Universal Robots PolyScope program: test2.v2objects.urp

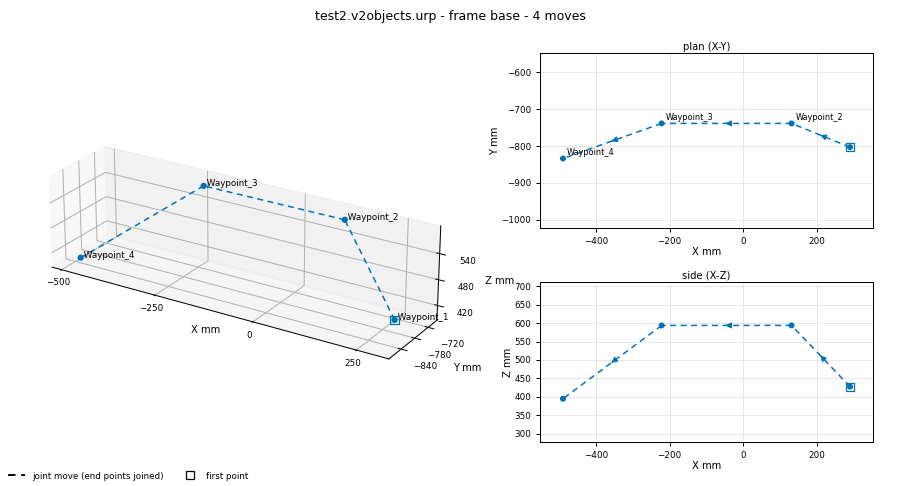
[picture p0: tool path of test2.v2objects.urp in frame base, 4 of 4 moves have a stored position in this frame; points joined in program order, loops and branches not executed]
Program test2.v2objects (installation=default directory=/programs/usbdisk/test 2_v2 createdIn=5.11.10.1010502 lastSavedIn=5.11.10.1010502 robotSerialNumber=20225201357)
Calibrated DH parameters: a=[-0.000097, -0.065329, -0.560646, 0.000001, -0.00004, 0]; d=[0.180831, -263.113709, 285.24385, -21.955837, 0.119737, 0.115719]; alpha=[1.571643, -0.002312, 0.004975, 1.569542, -1.570894, 0]; deltaTheta=[0, 1.463798, 5.013296, -0.193909, 0, 0]
Robot Program (runOnlyOnce=false)
  MoveJ speed 60 deg/s, acceleration 80 deg/s^2 (useActiveTCP=true) feature=Base
    Waypoint Waypoint_1: motionParameters(nextMotionTime=3); TCP in base x=289.597 y=-802.962 z=427.597 mm, rx=1.424 ry=0.8639 rz=-0.8474 rad; joints [100.839, -94.17, 117.361, -20.49, 99.76, 1.285] deg; TCP offset x=20.709 y=-1.468 z=254.962 mm, rx=-0.0022 ry=-0.0343 rz=-1.1076 rad
    Waypoint Waypoint_2: motionParameters(nextMotionTime=3); TCP in base x=130.852 y=-738.548 z=593.96 mm, rx=1.6172 ry=-0.3402 rz=0.3175 rad; joints [81.329, -110.965, 115.101, -1.443, 80.267, 87.015] deg
    Waypoint Waypoint_3: motionParameters(nextMotionTime=3); TCP in base x=-222.022 y=-738.536 z=593.824 mm, rx=1.6173 ry=-0.3402 rz=0.3176 rad; joints [34.019, -105.153, 111.263, -1.374, 33.032, 83.435] deg
    Waypoint Waypoint_4: motionParameters(nextMotionTime=3); TCP in base x=-489.837 y=-833.739 z=394.795 mm, rx=0.9699 ry=-1.6199 rz=1.5763 rad; joints [29.188, -77.516, 103.756, -22.876, 29.033, 180.614] deg
